FUNCTION F_Test1 : BOOL
VAR_INPUT
	stInput : ST_Test1;
END_VAR
VAR
END_VAR

F_Test1 := stInput.stBase.nTest1 < 100;
RETURN;

END_FUNCTION

(* stored: Version 1.1.0.1
   POU F_Test1: Id {e4b4edce-173d-4a99-bd33-931a37a8a1d4}, SpecialFunc None *)
